{attribute 'linkalways'} 
{attribute 'no_explicit_call' := 'This FB is a CLASS and must be accessed using methods or properties'}
{attribute 'enable_dynamic_creation'}
FUNCTION_BLOCK ChunkedRequestsMiddleware EXTENDS Middleware
VAR
	config : I_ChunkedRequestsMiddlewareConfig;
END_VAR

METHOD FB_init : BOOL
VAR_INPUT
	bInitRetains : BOOL; // if TRUE, the retain variables are initialized (warm start / cold start)
	bInCopyCode : BOOL;  // if TRUE, the instance afterwards gets moved into the copy code (online change)
	Config : I_ChunkedRequestsMiddlewareConfig;
END_VAR
THIS^.config := Config;
END_METHOD

METHOD PUBLIC Handle
VAR_INPUT
	Request : I_Request;
	Response : I_ServerResponse;
END_VAR
Next(Request, Response);
END_METHOD

METHOD PUBLIC UpdateConfig
VAR_INPUT
	Config : I_ChunkedRequestsMiddlewareConfig;
END_VAR
this^.config := Config;
END_METHOD

END_FUNCTION_BLOCK

(* stored: Version 1.1.0.1, ProductVersion 3.1.4024.12
   POU ChunkedRequestsMiddleware: Id {d274de03-f009-432b-96bd-8417c2bab972}, SpecialFunc None
   Folder Constructor: Id {c23e1ec0-1bb3-4041-baf7-c8106a918be7}
   Method FB_init: Id {34cb82f7-463b-49ef-a5d1-909c99be6633}
   Method Handle: Id {2756a409-70dc-4f3a-b4c9-8c97c902954c}
   Method UpdateConfig: Id {77c62bc4-deff-4f1f-b8c1-eee7a1bd6680} *)
